Staubli VAL3: getLibVersion.pgx

public program getLibVersion(string& x_sVersion[] (dimensions=1))
begin
  //-----------------------------------------------------------------------
  //Header begin
  //Description of program
  //  Retrieve version of the library.
  //
  //Output parameters
  //  string x_sVersion :
  //    role : version of the library
  //
  //Examples
  //  call getLibVersion(l_sLibVersion)
  //
  //History
  //  Creation : 19-05-08 - f.Rob
  //Header end
  //-----------------------------------------------------------------------

  x_sVersion=strVersion
end
